FUNCTION_BLOCK FB_AxisControl
VAR_INPUT
	Axis	: REFERENCE TO AXIS_REF;
END_VAR

VAR_OUTPUT
	AxisStatus : ST_AxisStatus;
	ErrorText : STRING;
END_VAR

VAR
	_MCMoveAbs	: MC_MoveAbsolute;
	_MCReset	: MC_Reset;
	_MCStop		: MC_Stop;
	_MCMoveVel	: MC_MoveVelocity;
	_MCPower	: MC_Power;
	_MCJog		: MC_Jog;
END_VAR

IF NOT __ISVALIDREF(Axis) THEN
	ErrorText := 'Axis Reference is Invalid.';
	RETURN;
ELSE
	ErrorText := '';
END_IF

_MCPower(Axis:= Axis,
			Enable:= TRUE,
			Enable_Positive:= TRUE,
			Enable_Negative:= TRUE,
			Override:= 100);
			
_MCReset(Axis:= Axis);
_MCStop(Axis:= Axis);
_MCMoveAbs(Axis:= Axis);
_MCMoveVel(Axis:= Axis);
_MCJog(Axis:= Axis);

Axis.ReadStatus();
AxisStatus := Axis.Status;

METHOD M_Jog
VAR_INPUT
	JogForward : BOOL;
	JogBackwards : BOOL;
	Mode : E_JogMode;
	Position : LREAL;
	Velocity : LREAL;
	Acceleration : LREAL;
	Deceleration : LREAL;
END_VAR

VAR_OUTPUT
	Done : BOOL;
	Error : BOOL;
	ErrorId : UDINT;
END_VAR
_MCJog.JogForward := JogForward;
_MCJog.JogBackwards := JogBackwards;
_MCJog.Mode := Mode;
_MCJog.Position := Position;
_MCJog.Velocity := Velocity;
_MCJog.Acceleration := Acceleration;
_MCJog.Deceleration := Deceleration;

Done := _MCJog.Done;
Error := _MCJog.Error;
ErrorId := _MCJog.ErrorId;
END_METHOD

METHOD M_MoveAbs
VAR_INPUT
	Execute : BOOL;
	Position : LREAL;
	Velocity : LREAL;
	Acceleration : LREAL;
	Deceleration : LREAL;
END_VAR

VAR_OUTPUT
	Done : BOOL;
	Error : BOOL;
END_VAR
_MCMoveAbs.Execute := Execute;
_MCMoveAbs.Position := Position;
_MCMoveAbs.Velocity := Velocity;
_MCMoveAbs.Acceleration := Acceleration;
_MCMoveAbs.Deceleration := Deceleration;

Done := _MCMoveAbs.Done;
Error := _MCMoveAbs.Error;
END_METHOD

METHOD M_MoveVel : BOOL
VAR_INPUT
	Execute : BOOL;
	Velocity : LREAL;
	Acceleration : LREAL;
	Deceleration : LREAL;
END_VAR
_MCMoveVel.Execute := Execute;
_MCMoveVel.Velocity := Velocity;
_MCMoveVel.Acceleration := Acceleration;
_MCMoveVel.Deceleration := Deceleration;
END_METHOD

METHOD M_Reset
VAR_INPUT
	Execute : BOOL;
END_VAR

VAR_OUTPUT
	Done : BOOL;
	Error : BOOL;
END_VAR
_MCReset.Execute := Execute;

Done := _MCReset.Done;
Error := _MCReset.Error;
END_METHOD

METHOD M_Stop
VAR_INPUT
	Execute : BOOL;
	Deceleration : LREAL;
END_VAR

VAR_OUTPUT
	Done : BOOL;
	Error : BOOL;
END_VAR
_MCStop.Execute := Execute;
_MCStop.Deceleration := Deceleration;

Done := _MCStop.Done;
Error := _MCStop.Error;
END_METHOD

END_FUNCTION_BLOCK

(* stored: Version 1.1.0.1, ProductVersion 3.1.4026.18
   POU FB_AxisControl: Id {28a42f80-195a-4223-a1bf-e623b7d6079c}, SpecialFunc None
   Method M_Jog: Id {dc88b92a-725e-4df4-aa19-7fa274329a3a}
   Method M_MoveAbs: Id {12c6fae0-35a4-42f7-a077-cdf0cbcaba8d}
   Method M_MoveVel: Id {2b358657-cee5-4620-ae42-419450a93b24}
   Method M_Reset: Id {73fb1eb2-f7fa-423b-ae99-c942ced73b28}
   Method M_Stop: Id {2df51e0d-c316-436a-9fe7-294a4bc52bdf} *)
